# EPICS autosave request: iocBoot/bkhDigiO.req
$(P):BO:SC:$(MOD):BIT$(N).DESC
$(P):BO:SC:$(MOD):BIT$(N).VAL
